PROGRAM POU_AxisMoveAbs
VAR
	fbAxis1MoveAbs:MC_MoveAbsolute;
	fbAxis1MoveAbs2:MC_MoveAbsolute;
	fbAxis2MoveAbs:MC_MoveAbsolute;
	fbAxis2MoveAbs2:MC_MoveAbsolute;
	fbAxis3MoveAbs:MC_MoveAbsolute;
	fbAxis3MoveAbs2:MC_MoveAbsolute;
	fbAxis4MoveAbs:MC_MoveAbsolute;
	fbAxis4MoveAbs2:MC_MoveAbsolute;
	fbAxis5MoveAbs:MC_MoveAbsolute;
	fbAxis5MoveAbs2:MC_MoveAbsolute;
	fbAxis6MoveAbs:MC_MoveAbsolute;
	fbAxis6MoveAbs2:MC_MoveAbsolute;
END_VAR

//Set Vertical Velocities
rAxisVelV:=0.5;
rAxis2Vel:=rAxisVelV;
rAxis4Vel:=rAxisVelV;
rAxis6Vel:=rAxisVelV;
//Set Horizontal Velocities
rAxisVelH:=1;
rAxis1Vel:=rAxisVelH;
rAxis3Vel:=rAxisVelH;
rAxis5Vel:=rAxisVelH;
//Create Each Move and Seccondary
fbAxis1MoveAbs(
	Axis:= Axis1, 
	Execute:= , 
	Position:=rAxis1Target , 
	Velocity:= rAxis1Vel, 
	Acceleration:= , 
	Deceleration:= , 
	Jerk:= , 
	BufferMode:=MC_BlendingLow , 
	Options:= , 
	Done=> , 
	Busy=> , 
	Active=> , 
	CommandAborted=> , 
	Error=> , 
	ErrorID=> );

fbAxis1MoveAbs2(
	Axis:= Axis1, 
	Execute:= , 
	Position:=rAxis1Target , 
	Velocity:=rAxis1Vel , 
	Acceleration:= , 
	Deceleration:= , 
	Jerk:= , 
	BufferMode:=MC_BlendingLow , 
	Options:= , 
	Done=> , 
	Busy=> , 
	Active=> , 
	CommandAborted=> , 
	Error=> , 
	ErrorID=> );
	
fbAxis2MoveAbs(
	Axis:= Axis2, 
	Execute:= , 
	Position:=rAxis2Target , 
	Velocity:= rAxis2Vel, 
	Acceleration:= , 
	Deceleration:= , 
	Jerk:= , 
	BufferMode:= MC_BlendingLow, 
	Options:= , 
	Done=> , 
	Busy=> , 
	Active=> , 
	CommandAborted=> , 
	Error=> , 
	ErrorID=> );
	
fbAxis2MoveAbs2(
	Axis:= Axis2, 
	Execute:= , 
	Position:=rAxis2Target , 
	Velocity:= rAxis2Vel, 
	Acceleration:= , 
	Deceleration:= , 
	Jerk:= , 
	BufferMode:=MC_BlendingLow , 
	Options:= , 
	Done=> , 
	Busy=> , 
	Active=> , 
	CommandAborted=> , 
	Error=> , 
	ErrorID=> );

fbAxis3MoveAbs(
	Axis:= Axis3, 
	Execute:= , 
	Position:=rAxis3Target , 
	Velocity:= rAxis3Vel, 
	Acceleration:= , 
	Deceleration:= , 
	Jerk:= , 
	BufferMode:=MC_BlendingLow , 
	Options:= , 
	Done=> , 
	Busy=> , 
	Active=> , 
	CommandAborted=> , 
	Error=> , 
	ErrorID=> );
	
fbAxis3MoveAbs2(
	Axis:= Axis3, 
	Execute:= , 
	Position:=rAxis3Target , 
	Velocity:= rAxis3Vel, 
	Acceleration:= , 
	Deceleration:= , 
	Jerk:= , 
	BufferMode:=MC_BlendingLow , 
	Options:= , 
	Done=> , 
	Busy=> , 
	Active=> , 
	CommandAborted=> , 
	Error=> , 
	ErrorID=> );
	
fbAxis4MoveAbs(
	Axis:= Axis4, 
	Execute:= , 
	Position:=rAxis4Target , 
	Velocity:= rAxis4Vel, 
	Acceleration:= , 
	Deceleration:= , 
	Jerk:= , 
	BufferMode:=MC_BlendingLow , 
	Options:= , 
	Done=> , 
	Busy=> , 
	Active=> , 
	CommandAborted=> , 
	Error=> , 
	ErrorID=> );
	
fbAxis4MoveAbs2(
	Axis:= Axis4, 
	Execute:= , 
	Position:=rAxis4Target , 
	Velocity:= rAxis4Vel, 
	Acceleration:= , 
	Deceleration:= , 
	Jerk:= , 
	BufferMode:=MC_BlendingLow , 
	Options:= , 
	Done=> , 
	Busy=> , 
	Active=> , 
	CommandAborted=> , 
	Error=> , 
	ErrorID=> );
	
fbAxis5MoveAbs(
	Axis:= Axis5, 
	Execute:= , 
	Position:=rAxis5Target , 
	Velocity:=rAxis5Vel , 
	Acceleration:= , 
	Deceleration:= , 
	Jerk:= , 
	BufferMode:=MC_BlendingLow , 
	Options:= , 
	Done=> , 
	Busy=> , 
	Active=> , 
	CommandAborted=> , 
	Error=> , 
	ErrorID=> );
	
fbAxis5MoveAbs2(
	Axis:= Axis5, 
	Execute:= , 
	Position:=rAxis5Target , 
	Velocity:= rAxis5Vel, 
	Acceleration:= , 
	Deceleration:= , 
	Jerk:= , 
	BufferMode:=MC_BlendingLow , 
	Options:= , 
	Done=> , 
	Busy=> , 
	Active=> , 
	CommandAborted=> , 
	Error=> , 
	ErrorID=> );
	
fbAxis6MoveAbs(
	Axis:= Axis6, 
	Execute:= , 
	Position:=rAxis6Target , 
	Velocity:= rAxis6Vel, 
	Acceleration:= , 
	Deceleration:= , 
	Jerk:= , 
	BufferMode:=MC_BlendingLow , 
	Options:= , 
	Done=> , 
	Busy=> , 
	Active=> , 
	CommandAborted=> , 
	Error=> , 
	ErrorID=> );
	
fbAxis6MoveAbs2(
	Axis:= Axis6, 
	Execute:= , 
	Position:=rAxis6Target , 
	Velocity:= rAxis6Vel, 
	Acceleration:= , 
	Deceleration:= , 
	Jerk:= , 
	BufferMode:= MC_BlendingLow, 
	Options:= , 
	Done=> , 
	Busy=> , 
	Active=> , 
	CommandAborted=> , 
	Error=> , 
	ErrorID=> );
	


	IF bAxis1Enable	THEN
		IF bAxis1MoveABS THEN
			IF fbAxis1MoveAbs.Busy THEN
				IF fbAxis1MoveAbs2.Busy	THEN
					;
				ELSE
					fbAxis1MoveAbs2.Execute:=TRUE;
					bAxis1MoveAbs:=FALSE;
				END_IF
			ELSE
				fbAxis1MoveAbs.Execute:=TRUE;
				bAxis1MoveAbs:=FALSE;
			END_IF
		ELSIF fbAxis1MoveAbs.Done THEN
			bAxis1MoveAbs:=FALSE;
			fbAxis1MoveAbs.Execute:=FALSE;
		ELSIF fbAxis1MoveAbs2.Done THEN
			bAxis1MoveAbs:=FALSE;
			fbAxis1MoveAbs2.Execute:=FALSE;
		END_IF
	ELSE 
		fbAxis1MoveAbs2.Execute:=FALSE;
		fbAxis1MoveAbs.Execute:=FALSE;
	END_IF
	
	IF bAxis2Enable THEN
		IF bAxis2MoveABS THEN
			IF fbAxis2MoveAbs.Busy THEN
				IF fbAxis2MoveAbs2.Busy THEN
				;
				ELSE	
					fbAxis2MoveAbs2.Execute:=TRUE;
					bAxis2MoveAbs:=FALSE;
				END_IF
			ELSE
				fbAxis2MoveAbs.Execute:=TRUE;
				bAxis2MoveAbs:=FALSE;
			END_IF
		ELSIF fbAxis2MoveAbs.Done THEN
			bAxis2MoveAbs:=FALSE;
			fbAxis2MoveAbs.Execute:=FALSE;
		ELSIF fbAxis2MoveAbs2.Done THEN
			bAxis2MoveAbs:=FALSE;
			fbAxis2MoveAbs2.Execute:=FALSE;
		END_IF
	ELSE 
		fbAxis2MoveAbs2.Execute:=FALSE;
		fbAxis2MoveAbs.Execute:=FALSE;
	END_IF
	
	IF bAxis3Enable THEN
		IF bAxis3MoveABS THEN
			IF fbAxis3MoveAbs.Busy THEN
				IF fbAxis3MoveAbs2.Busy THEN
					;
				ELSE
					fbAxis3MoveAbs2.Execute:=TRUE;
					bAxis3MoveAbs:=FALSE;
				END_IF
			ELSE
				fbAxis3MoveAbs.Execute:=TRUE;
				bAxis3MoveAbs:=FALSE;
			END_IF
		ELSIF fbAxis3MoveAbs.Done THEN
			bAxis3MoveAbs:=FALSE;
			fbAxis3MoveAbs.Execute:=FALSE;
		ELSIF fbAxis3MoveAbs2.Done THEN
			bAxis3MoveAbs:=FALSE;
			fbAxis3MoveAbs2.Execute:=FALSE;
		END_IF
	ELSE 
		fbAxis3MoveAbs2.Execute:=FALSE;
		fbAxis3MoveAbs.Execute:=FALSE;
	END_IF
	
	IF bAxis4Enable THEN
		IF bAxis4MoveABS THEN
			IF fbAxis4MoveAbs.Busy THEN
				IF fbAxis4MoveAbs2.Busy THEN
					;
				ELSE
					fbAxis4MoveAbs2.Execute:=TRUE;
					bAxis4MoveAbs:=FALSE;
				END_IF
			ELSE
				fbAxis4MoveAbs.Execute:=TRUE;
				bAxis4MoveAbs:=FALSE;
			END_IF
		ELSIF fbAxis4MoveAbs.Done THEN
			bAxis4MoveAbs:=FALSE;
			fbAxis4MoveAbs.Execute:=FALSE;
		ELSIF fbAxis4MoveAbs2.Done THEN
			bAxis4MoveAbs:=FALSE;
			fbAxis4MoveAbs2.Execute:=FALSE;
			
		END_IF		
	ELSE 
		fbAxis4MoveAbs2.Execute:=FALSE;
		fbAxis4MoveAbs.Execute:=FALSE;
	END_IF
	
	IF bAxis5Enable THEN
		IF bAxis5MoveABS THEN
			IF fbAxis5MoveAbs.Busy THEN
				IF fbAxis5MoveAbs2.Busy THEN
					;
				ELSE
					fbAxis5MoveAbs2.Execute:=TRUE;
					bAxis5MoveAbs:=FALSE;
				END_IF
			ELSE
				fbAxis5MoveAbs.Execute:=TRUE;
				bAxis5MoveAbs:=FALSE;
			END_IF
		ELSIF fbAxis5MoveAbs.Done THEN
			bAxis5MoveAbs:=FALSE;
			fbAxis5MoveAbs.Execute:=FALSE;
		ELSIF fbAxis5MoveAbs2.Done THEN
			bAxis5MoveAbs:=FALSE;
			fbAxis5MoveAbs2.Execute:=FALSE;
		END_IF
	ELSE 
		fbAxis5MoveAbs2.Execute:=FALSE;
		fbAxis5MoveAbs.Execute:=FALSE;
	END_IF
	
	IF bAxis6Enable THEN
		IF bAxis6MoveABS THEN
			IF fbAxis6MoveAbs.Busy THEN
				IF fbAxis6MoveAbs2.Busy THEN
					;
				ELSE
					fbAxis6MoveAbs2.Execute:=TRUE;
					bAxis6MoveAbs:=FALSE;
				END_IF
			ELSE
				fbAxis6MoveAbs.Execute:=TRUE;
				bAxis6MoveAbs:=FALSE;
			END_IF
		ELSIF fbAxis6MoveAbs.Done THEN
			bAxis6MoveAbs:=FALSE;
			fbAxis6MoveAbs.Execute:=FALSE;
		ELSIF fbAxis6MoveAbs2.Done THEN
			bAxis6MoveAbs:=FALSE;
			fbAxis6MoveAbs2.Execute:=FALSE;
		ELSE 
			fbAxis6MoveAbs2.Execute:=FALSE;
			fbAxis6MoveAbs.Execute:=FALSE;
		END_IF
	ELSE 
		fbAxis6MoveAbs2.Execute:=FALSE;
		fbAxis6MoveAbs.Execute:=FALSE;
	END_IF

END_PROGRAM

(* stored: Version 1.1.0.1, ProductVersion 3.1.4022.18
   POU POU_AxisMoveAbs: Id {5b341b12-8db7-4b40-b8e2-bfd744022721}, SpecialFunc None *)
